PROGRAM P_ControlBlock
VAR
	fbControlBlock : c_FB_ControlBlockWithMonito;
	fbMotionRef : FB_MotionReference;
	fbJoyRef : FB_Joystick_2;
	fbClock : FB_Clock;
	fbInitialPos : FB_InitialPos;
	fbInitialPa : FB_InitialPressure;
	fbInitialPb : FB_InitialPressure;
	fbInitialPs : FB_InitialPressure;
	InitialPa : LREAL;
	
END_VAR

fbClock(
	bStart := G_Inputs.bStartButton,
	bStop := G_Inputs.bStopButton,
	fCycleTime :=0.001
);

fbInitialPos(
	bEnable := (G_Work.eStatus = E_Status.Running),
	fCurrentPos := G_Sensors.fPistonPosition,
);

fbInitialPa(
	bEnable := (G_Work.eStatus = E_Status.Running),
	fCurrentPressure := G_Sensors.fPressurePistonSide,
);

fbInitialPb(
	bEnable := (G_Work.eStatus = E_Status.Running),
	fCurrentPressure := G_Sensors.fPressureRodSide,
);

fbInitialPs(
	bEnable := (G_Work.eStatus = E_Status.Running),
	fCurrentPressure := G_Sensors.fPressureSupply,
);

//InitialPa := fbInitialPa.fCurrentPressure;

IF (G_Work.eMode = E_Mode.Auto) THEN
	
	G_OPC_UA.fXRef := fbMotionRef.fPositionReference_m;
	G_OPC_UA.fXDotRef := fbMotionRef.fVelocityReference_ms;
	
	fbMotionRef(
		fStartPosition_m := fbInitialPos.fInitialPos,
		fStartVelocity_m := 0,
		fPositionSetpoint_ms := 0.3,
		fVelocitySetpoint_m := G_Parameter.fMaxSpeed,
		fTimeBeforeStarting_s := 1,
		fRampTime_s := 1,
		fHoldPositionTime_s := 1,
		fClock_s:= fbClock.fTime,
		bEnable:= G_Inputs.bStartButton
	);
	
	

	
	fbControlBlock(
		ssMethodType := BOOL_TO_SINT(G_Work.eStatus = E_Status.Running),
		bEnablePID := G_Parameter.bEnablePID,
		bEnableU := G_Parameter.bEnableU,
		
		X_real:= G_Sensors.fPistonPosition,
		X_dot := fbMotionRef.fVelocityReference_ms,
		X := fbMotionRef.fPositionReference_m,
		Pa := G_Sensors.fPressurePistonSide, 
		Pb := G_Sensors.fPressureRodSide,
		Ps := G_Sensors.fPressureSupply,
		
		InitialPs := fbInitialPs.fCurrentPressure,
		InitialPa := InitialPa,
		InitialPb := fbInitialPb.fCurrentPressure,
		
		U	=> G_Work.fControlOutputNormalized
	);

ELSIF (G_Work.eMode = E_Mode.Manual) THEN

	G_OPC_UA.fXRef := fbJoyRef.fPositionReferance_m;
	G_OPC_UA.fXDotRef := fbJoyRef.fVelocityReferance_ms;
	
	fbJoyRef(
		ssMethodType := BOOL_TO_SINT(G_Work.eStatus = E_Status.Running),
		Joystick := G_Sensors.fJoystickY,
		XInital := fbInitialPos.fInitialPos,
	);

	
	fbControlBlock(
	ssMethodType := BOOL_TO_SINT(G_Work.eStatus = E_Status.Running),
	bEnablePID := G_Parameter.bEnablePID,
	bEnableU := G_Parameter.bEnableU,
		
	X_real:= G_Sensors.fPistonPosition,
	X_dot := fbJoyRef.fVelocityReferance_ms,
	X := fbJoyRef.fPositionReferance_m,
	Pa:= G_Sensors.fPressurePistonSide, 
	Pb := G_Sensors.fPressureRodSide,
	Ps:= G_Sensors.fPressureSupply,
	
	InitialPs := fbInitialPs.fCurrentPressure,
	InitialPa := fbInitialPa.fCurrentPressure,
	InitialPb := fbInitialPb.fCurrentPressure,
	
	U	=> G_Work.fControlOutputNormalized
	);
	
END_IF

END_PROGRAM

(* stored: Version 1.1.0.1, ProductVersion 3.1.4024.12
   POU P_ControlBlock: Id {1c742f8d-99bf-4aa1-ba99-fa370ccce2ab}, SpecialFunc None *)
